// SIMATIC S7-200 project (STEP 7-Micro/WIN), CPU 226 REL 02.01

ORGANIZATION_BLOCK 主程序:OB1
TITLE=程序注释
BEGIN
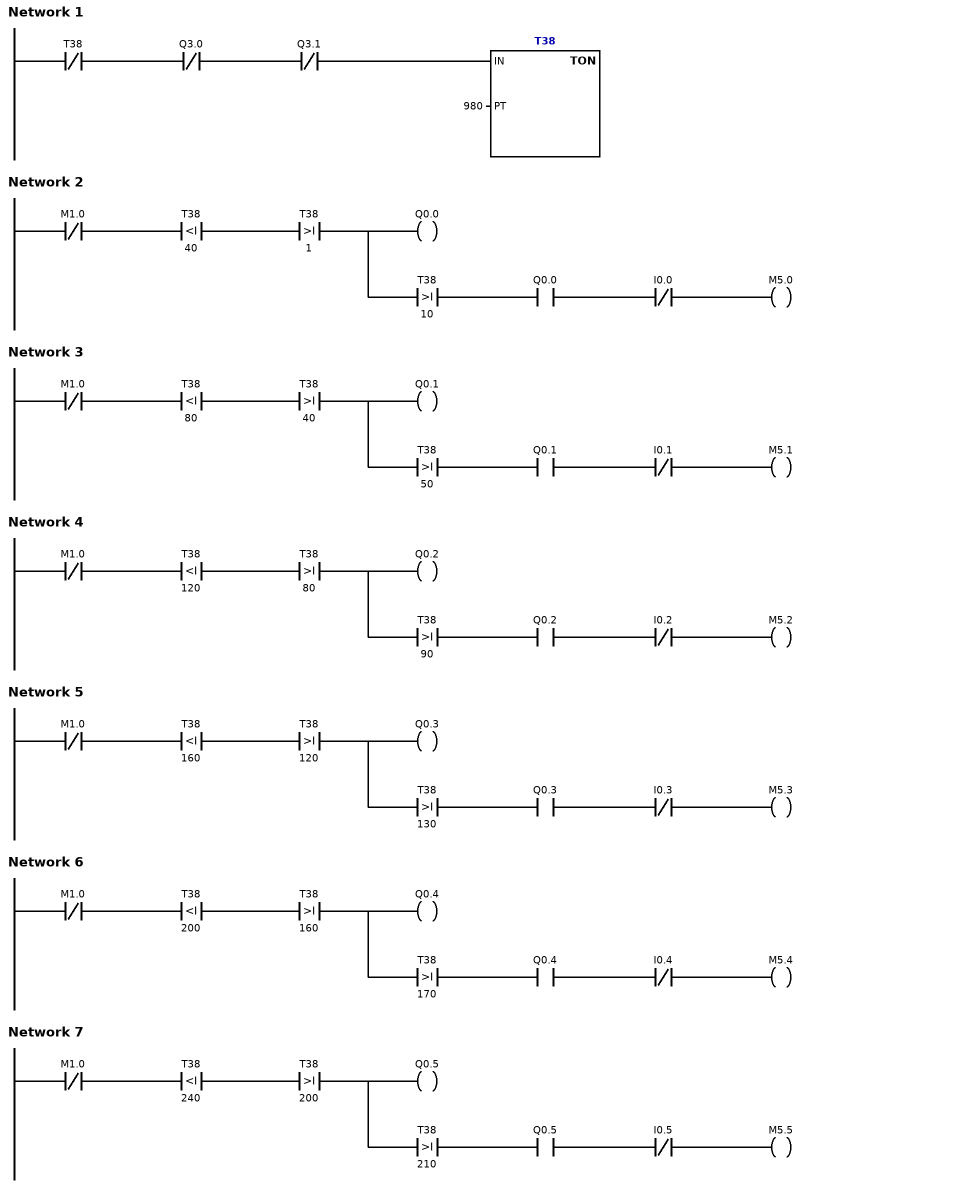
Network 1
LDN    T38
AN     Q3.0
AN     Q3.1
TON    T38, 980
Network 2
LDN    M1.0
AW<    T38, 40
AW>    T38, 1
=      Q0.0
AW>    T38, 10
A      Q0.0
AN     I0.0
=      M5.0
Network 3
LDN    M1.0
AW<    T38, 80
AW>    T38, 40
=      Q0.1
AW>    T38, 50
A      Q0.1
AN     I0.1
=      M5.1
Network 4
LDN    M1.0
AW<    T38, 120
AW>    T38, 80
=      Q0.2
AW>    T38, 90
A      Q0.2
AN     I0.2
=      M5.2
Network 5
LDN    M1.0
AW<    T38, 160
AW>    T38, 120
=      Q0.3
AW>    T38, 130
A      Q0.3
AN     I0.3
=      M5.3
Network 6
LDN    M1.0
AW<    T38, 200
AW>    T38, 160
=      Q0.4
AW>    T38, 170
A      Q0.4
AN     I0.4
=      M5.4
Network 7
LDN    M1.0
AW<    T38, 240
AW>    T38, 200
=      Q0.5
AW>    T38, 210
A      Q0.5
AN     I0.5
=      M5.5
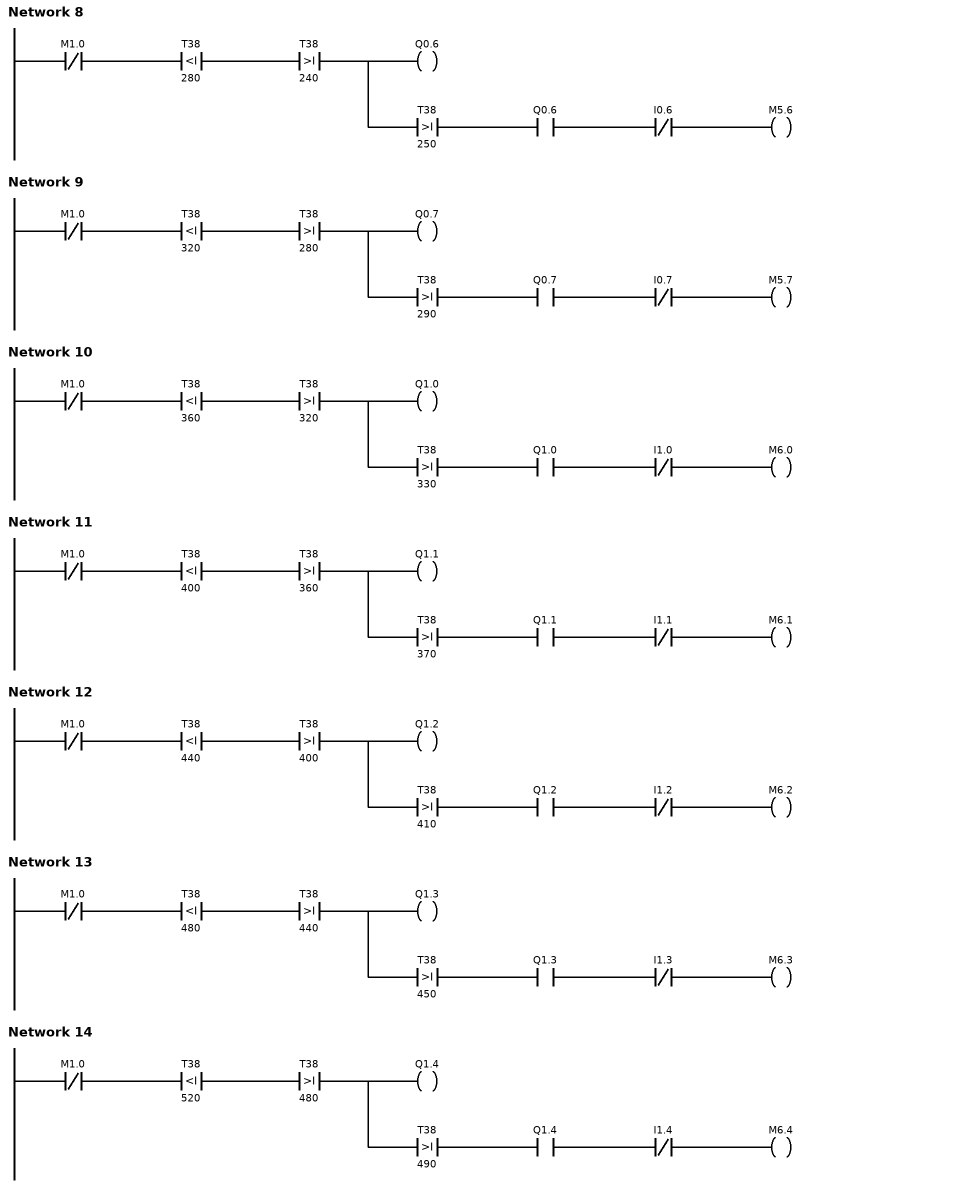
Network 8
LDN    M1.0
AW<    T38, 280
AW>    T38, 240
=      Q0.6
AW>    T38, 250
A      Q0.6
AN     I0.6
=      M5.6
Network 9
LDN    M1.0
AW<    T38, 320
AW>    T38, 280
=      Q0.7
AW>    T38, 290
A      Q0.7
AN     I0.7
=      M5.7
Network 10
LDN    M1.0
AW<    T38, 360
AW>    T38, 320
=      Q1.0
AW>    T38, 330
A      Q1.0
AN     I1.0
=      M6.0
Network 11
LDN    M1.0
AW<    T38, 400
AW>    T38, 360
=      Q1.1
AW>    T38, 370
A      Q1.1
AN     I1.1
=      M6.1
Network 12
LDN    M1.0
AW<    T38, 440
AW>    T38, 400
=      Q1.2
AW>    T38, 410
A      Q1.2
AN     I1.2
=      M6.2
Network 13
LDN    M1.0
AW<    T38, 480
AW>    T38, 440
=      Q1.3
AW>    T38, 450
A      Q1.3
AN     I1.3
=      M6.3
Network 14
LDN    M1.0
AW<    T38, 520
AW>    T38, 480
=      Q1.4
AW>    T38, 490
A      Q1.4
AN     I1.4
=      M6.4
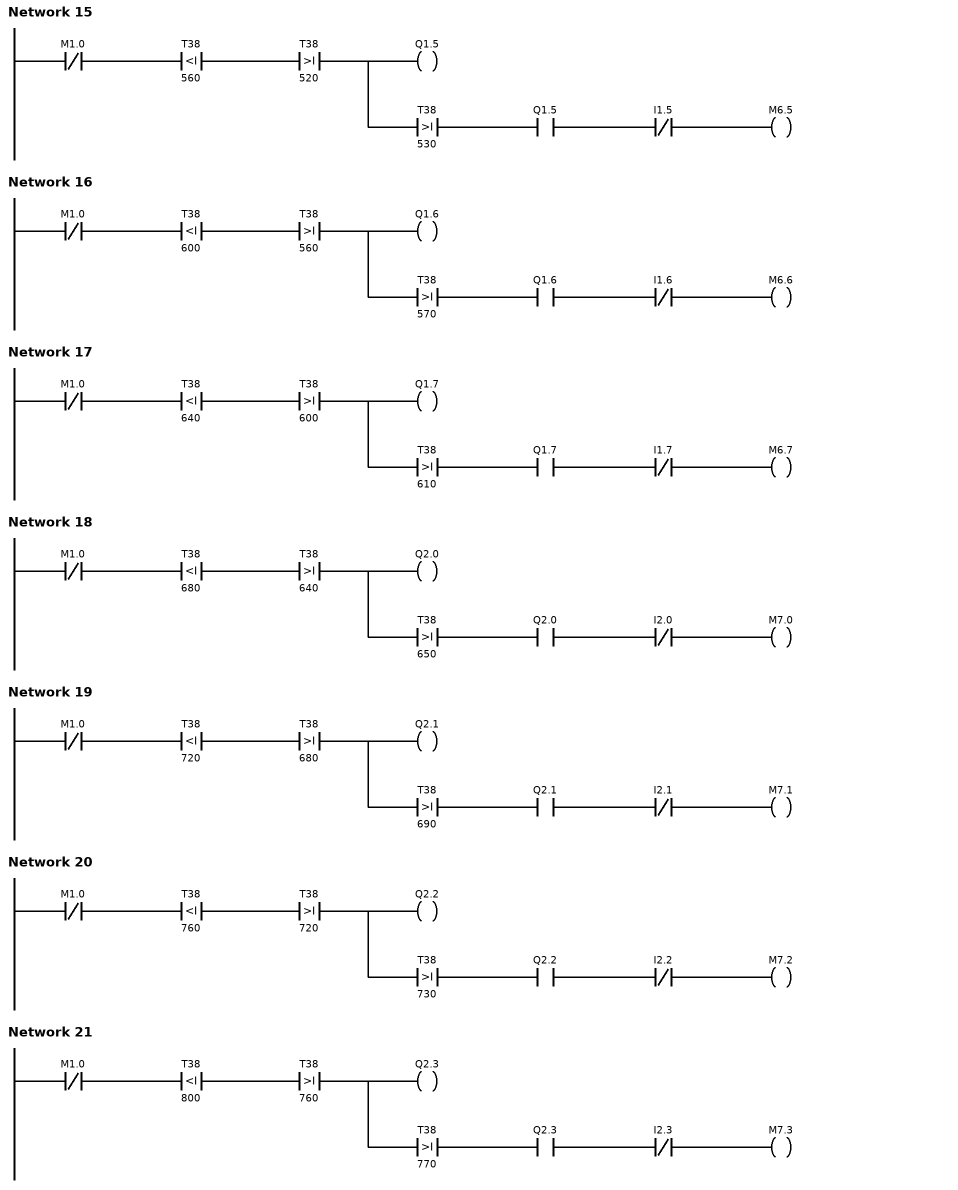
Network 15
LDN    M1.0
AW<    T38, 560
AW>    T38, 520
=      Q1.5
AW>    T38, 530
A      Q1.5
AN     I1.5
=      M6.5
Network 16
LDN    M1.0
AW<    T38, 600
AW>    T38, 560
=      Q1.6
AW>    T38, 570
A      Q1.6
AN     I1.6
=      M6.6
Network 17
LDN    M1.0
AW<    T38, 640
AW>    T38, 600
=      Q1.7
AW>    T38, 610
A      Q1.7
AN     I1.7
=      M6.7
Network 18
LDN    M1.0
AW<    T38, 680
AW>    T38, 640
=      Q2.0
AW>    T38, 650
A      Q2.0
AN     I2.0
=      M7.0
Network 19
LDN    M1.0
AW<    T38, 720
AW>    T38, 680
=      Q2.1
AW>    T38, 690
A      Q2.1
AN     I2.1
=      M7.1
Network 20
LDN    M1.0
AW<    T38, 760
AW>    T38, 720
=      Q2.2
AW>    T38, 730
A      Q2.2
AN     I2.2
=      M7.2
Network 21
LDN    M1.0
AW<    T38, 800
AW>    T38, 760
=      Q2.3
AW>    T38, 770
A      Q2.3
AN     I2.3
=      M7.3
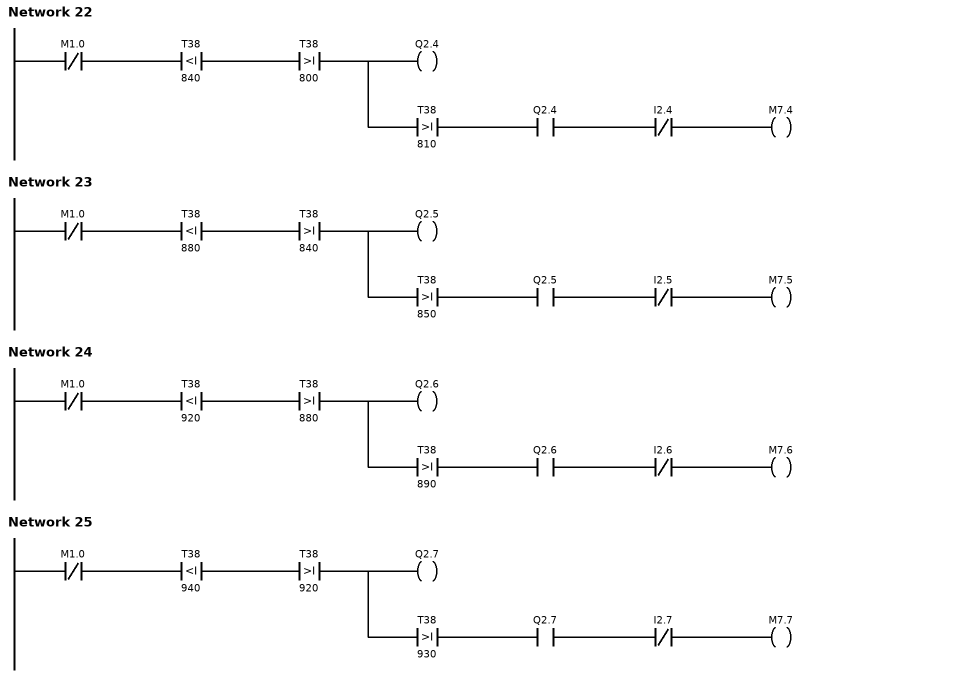
Network 22
LDN    M1.0
AW<    T38, 840
AW>    T38, 800
=      Q2.4
AW>    T38, 810
A      Q2.4
AN     I2.4
=      M7.4
Network 23
LDN    M1.0
AW<    T38, 880
AW>    T38, 840
=      Q2.5
AW>    T38, 850
A      Q2.5
AN     I2.5
=      M7.5
Network 24
LDN    M1.0
AW<    T38, 920
AW>    T38, 880
=      Q2.6
AW>    T38, 890
A      Q2.6
AN     I2.6
=      M7.6
Network 25
LDN    M1.0
AW<    T38, 940
AW>    T38, 920
=      Q2.7
AW>    T38, 930
A      Q2.7
AN     I2.7
=      M7.7
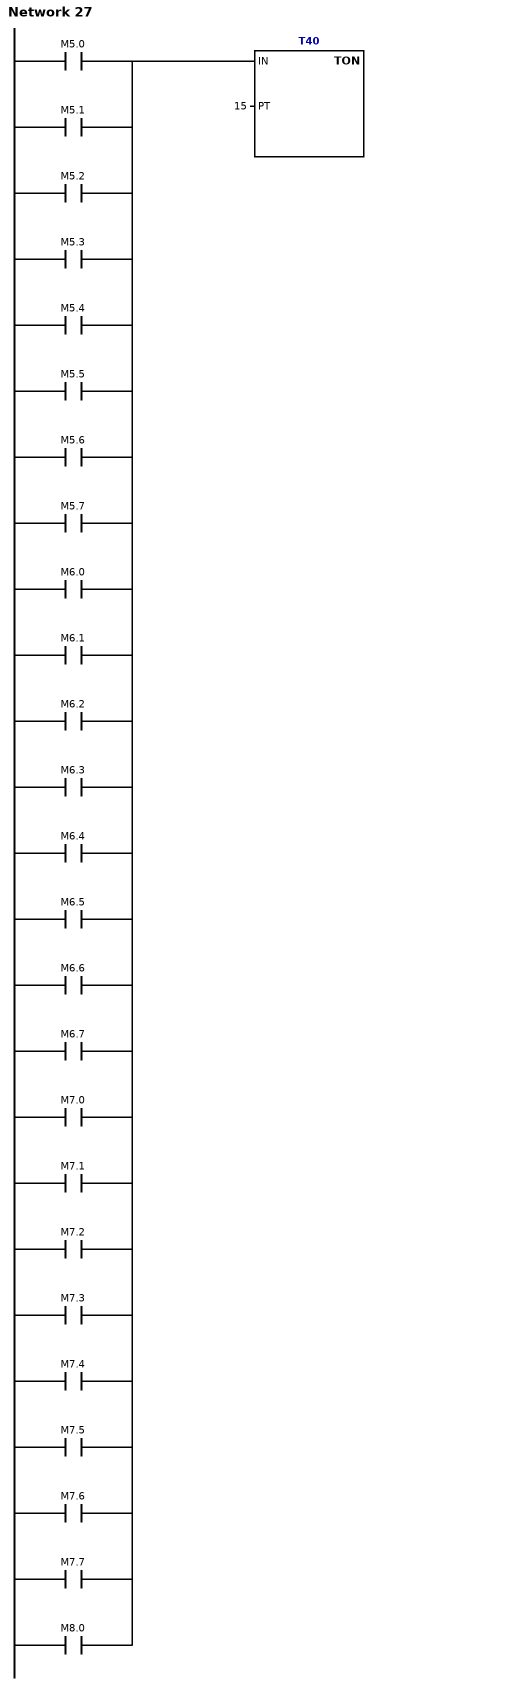
Network 27
LD     M5.0
O      M5.1
O      M5.2
O      M5.3
O      M5.4
O      M5.5
O      M5.6
O      M5.7
O      M6.0
O      M6.1
O      M6.2
O      M6.3
O      M6.4
O      M6.5
O      M6.6
O      M6.7
O      M7.0
O      M7.1
O      M7.2
O      M7.3
O      M7.4
O      M7.5
O      M7.6
O      M7.7
O      M8.0
TON    T40, 15
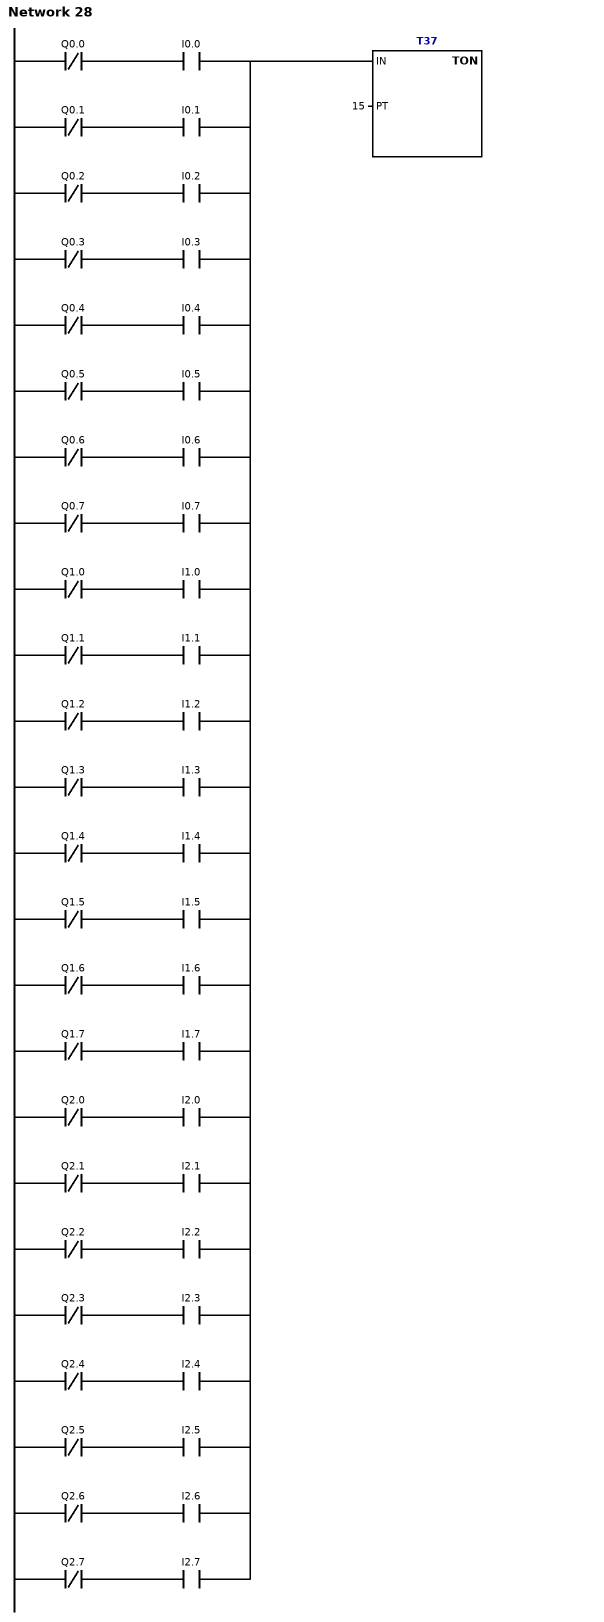
Network 28
LDN    Q0.0
A      I0.0
LDN    Q0.1
A      I0.1
OLD
LDN    Q0.2
A      I0.2
OLD
LDN    Q0.3
A      I0.3
OLD
LDN    Q0.4
A      I0.4
OLD
LDN    Q0.5
A      I0.5
OLD
LDN    Q0.6
A      I0.6
OLD
LDN    Q0.7
A      I0.7
OLD
LDN    Q1.0
A      I1.0
OLD
LDN    Q1.1
A      I1.1
OLD
LDN    Q1.2
A      I1.2
OLD
LDN    Q1.3
A      I1.3
OLD
LDN    Q1.4
A      I1.4
OLD
LDN    Q1.5
A      I1.5
OLD
LDN    Q1.6
A      I1.6
OLD
LDN    Q1.7
A      I1.7
OLD
LDN    Q2.0
A      I2.0
OLD
LDN    Q2.1
A      I2.1
OLD
LDN    Q2.2
A      I2.2
OLD
LDN    Q2.3
A      I2.3
OLD
LDN    Q2.4
A      I2.4
OLD
LDN    Q2.5
A      I2.5
OLD
LDN    Q2.6
A      I2.6
OLD
LDN    Q2.7
A      I2.7
OLD
TON    T37, 15
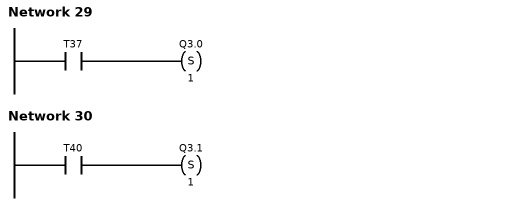
Network 29
LD     T37
S      Q3.0, 1
Network 30
LD     T40
S      Q3.1, 1
END_ORGANIZATION_BLOCK
